(* IEC 61131-3 sources: eCockpitGit/test_project/src/%F%00 Library/%F%Common Functions/%F%String/%F%Big Input/%F%Concat, 9 files *)

(* ---- %POU%FU_sConcat10BI.st ---- *)
//This functions combines ten strings
//This is the big input version which means any size string can be inputted, but only string variables will be accepted
//It is also faster on bigger strings
// |**Version**|**Author**| **Date** |**Changes**
// | 1         | NSN      | 05-02-19 | Creation
// | 2         | NSN      | 14-10-21 | Changed to pointer based
FUNCTION FU_sConcat10BI : STRING(255)
VAR_INPUT
	s1			:POINTER TO EASCII;			//Input String1
	s2			:POINTER TO EASCII;			//Input String2
	s3			:POINTER TO EASCII;			//Input String3
	s4			:POINTER TO EASCII;			//Input String4
	s5			:POINTER TO EASCII;			//Input String5
	s6			:POINTER TO EASCII;			//Input String6
	s7			:POINTER TO EASCII;			//Input String7
	s8			:POINTER TO EASCII;			//Input String8
	s9			:POINTER TO EASCII;			//Input String9
	s10			:POINTER TO EASCII;			//Input String10
END_VAR
(*%!%__DELIMITER__%!%*)
FU_sConcat10BIBO(sOut:=ADR(FU_sConcat10BI),s1:=s1,s2:=s2,s3:=s3,s4:=s4,s5:=s5,s6:=s6,s7:=s7,s8:=s8,s9:=s9,s10:=s10,wOutSize:=255);

(* ---- %POU%FU_sConcat3BI.st ---- *)
//This functions combines three strings
//This is the big input version which means any size string can be inputted, but only string variables will be accepted
//It is also faster on bigger strings
// |**Version**|**Author**| **Date** |**Changes**
// | 1         | NSN      | 05-02-19 | Creation
// | 2         | NSN      | 14-10-21 | Changed to pointer based
FUNCTION FU_sConcat3BI : STRING(255)
VAR_INPUT
	s1			:POINTER TO EASCII;						//Input String1
	s2			:POINTER TO EASCII;						//Input String2
	s3			:POINTER TO EASCII;						//Input String3
END_VAR
(*%!%__DELIMITER__%!%*)
FU_sConcat3BIBO(sOut:=ADR(FU_sConcat3BI),s1:=s1,s2:=s2,s3:=s3,wOutSize:=255);

(* ---- %POU%FU_sConcat4BI.st ---- *)
//This functions combines four strings
//This is the big input version which means any size string can be inputted, but only string variables will be accepted
//It is also faster on bigger strings
// |**Version**|**Author**| **Date** |**Changes**
// | 1         | NSN      | 05-02-19 | Creation
// | 2         | NSN      | 14-10-21 | Changed to pointer based
FUNCTION FU_sConcat4BI : STRING(255)
VAR_INPUT
	s1			:POINTER TO EASCII;			//Input String1
	s2			:POINTER TO EASCII;			//Input String2
	s3			:POINTER TO EASCII;			//Input String3
	s4			:POINTER TO EASCII;			//Input String4
END_VAR
(*%!%__DELIMITER__%!%*)
FU_sConcat4BIBO(sOut:=ADR(FU_sConcat4BI),s1:=s1,s2:=s2,s3:=s3,s4:=s4,wOutSize:=255);

(* ---- %POU%FU_sConcat5BI.st ---- *)
//This functions combines five strings
//This is the big input version which means any size string can be inputted, but only string variables will be accepted
//It is also faster on bigger strings
// |**Version**|**Author**| **Date** |**Changes**
// | 1         | NSN      | 05-02-19 | Creation
// | 2         | NSN      | 14-10-21 | Changed to pointer based
FUNCTION FU_sConcat5BI : STRING(255)
VAR_INPUT
	s1			:POINTER TO EASCII;			//Input String1
	s2			:POINTER TO EASCII;			//Input String2
	s3			:POINTER TO EASCII;			//Input String3
	s4			:POINTER TO EASCII;			//Input String4
	s5			:POINTER TO EASCII;			//Input String5
END_VAR
(*%!%__DELIMITER__%!%*)
FU_sConcat5BIBO(sOut:=ADR(FU_sConcat5BI),s1:=s1,s2:=s2,s3:=s3,s4:=s4,s5:=s5,wOutSize:=255);

(* ---- %POU%FU_sConcat6BI.st ---- *)
//This functions combines six strings
//This is the big input version which means any size string can be inputted, but only string variables will be accepted
//It is also faster on bigger strings
// |**Version**|**Author**| **Date** |**Changes**
// | 1         | NSN      | 05-02-19 | Creation
// | 2         | NSN      | 14-10-21 | Changed to pointer based
FUNCTION FU_sConcat6BI : STRING(255)
VAR_INPUT
	s1			:POINTER TO EASCII;			//Input String1
	s2			:POINTER TO EASCII;			//Input String2
	s3			:POINTER TO EASCII;			//Input String3
	s4			:POINTER TO EASCII;			//Input String4
	s5			:POINTER TO EASCII;			//Input String5
	s6			:POINTER TO EASCII;			//Input String6
END_VAR
(*%!%__DELIMITER__%!%*)
FU_sConcat6BIBO(sOut:=ADR(FU_sConcat6BI),s1:=s1,s2:=s2,s3:=s3,s4:=s4,s5:=s5,s6:=s6,wOutSize:=255);

(* ---- %POU%FU_sConcat7BI.st ---- *)
//This functions combines seven strings
//This is the big input version which means any size string can be inputted, but only string variables will be accepted
//It is also faster on bigger strings
// |**Version**|**Author**| **Date** |**Changes**
// | 1         | NSN      | 05-02-19 | Creation
// | 2         | NSN      | 14-10-21 | Changed to pointer based
FUNCTION FU_sConcat7BI : STRING(255)
VAR_INPUT
	s1			:POINTER TO EASCII;			//Input String1
	s2			:POINTER TO EASCII;			//Input String2
	s3			:POINTER TO EASCII;			//Input String3
	s4			:POINTER TO EASCII;			//Input String4
	s5			:POINTER TO EASCII;			//Input String5
	s6			:POINTER TO EASCII;			//Input String6
	s7			:POINTER TO EASCII;			//Input String7
END_VAR
(*%!%__DELIMITER__%!%*)
FU_sConcat7BIBO(sOut:=ADR(FU_sConcat7BI),s1:=s1,s2:=s2,s3:=s3,s4:=s4,s5:=s5,s6:=s6,s7:=s7,wOutSize:=255);

(* ---- %POU%FU_sConcat8BI.st ---- *)
//This functions combines nine strings
//This is the big input version which means any size string can be inputted, but only string variables will be accepted
//It is also faster on bigger strings
// |**Version**|**Author**| **Date** |**Changes**
// | 1         | NSN      | 05-02-19 | Creation
// | 2         | NSN      | 14-10-21 | Changed to pointer based
FUNCTION FU_sConcat8BI : STRING(255)
VAR_INPUT
	s1			:POINTER TO EASCII;			//Input String1
	s2			:POINTER TO EASCII;			//Input String2
	s3			:POINTER TO EASCII;			//Input String3
	s4			:POINTER TO EASCII;			//Input String4
	s5			:POINTER TO EASCII;			//Input String5
	s6			:POINTER TO EASCII;			//Input String6
	s7			:POINTER TO EASCII;			//Input String7
	s8			:POINTER TO EASCII;			//Input String8
END_VAR
(*%!%__DELIMITER__%!%*)
FU_sConcat8BIBO(sOut:=ADR(FU_sConcat8BI),s1:=s1,s2:=s2,s3:=s3,s4:=s4,s5:=s5,s6:=s6,s7:=s7,s8:=s8,wOutSize:=255);

(* ---- %POU%FU_sConcat9BI.st ---- *)
//This functions combines nine strings
//This is the big input version which means any size string can be inputted, but only string variables will be accepted
//It is also faster on bigger strings
// |**Version**|**Author**| **Date** |**Changes**
// | 1         | NSN      | 05-02-19 | Creation
// | 2         | NSN      | 14-10-21 | Changed to pointer based
FUNCTION FU_sConcat9BI : STRING(255)
VAR_INPUT
	s1			:POINTER TO EASCII;			//Input String1
	s2			:POINTER TO EASCII;			//Input String2
	s3			:POINTER TO EASCII;			//Input String3
	s4			:POINTER TO EASCII;			//Input String4
	s5			:POINTER TO EASCII;			//Input String5
	s6			:POINTER TO EASCII;			//Input String6
	s7			:POINTER TO EASCII;			//Input String7
	s8			:POINTER TO EASCII;			//Input String8
	s9			:POINTER TO EASCII;			//Input String9
END_VAR
(*%!%__DELIMITER__%!%*)
FU_sConcat9BIBO(sOut:=ADR(FU_sConcat9BI),s1:=s1,s2:=s2,s3:=s3,s4:=s4,s5:=s5,s6:=s6,s7:=s7,s8:=s8,s9:=s9,wOutSize:=255);

(* ---- %POU%FU_sConcatBI.st ---- *)
//This functions combines two strings
//This is the big input version which means any size string can be inputted, but only string variables will be accepted
//It is also faster on bigger strings
// |**Version**|**Author**| **Date** |**Changes**
// | 1         | NSN      | 05-02-19 | Creation
// | 2         | NSN      | 14-10-21 | Changed to pointer based
FUNCTION FU_sConcatBI : STRING(255)
VAR_INPUT
	s1			:POINTER TO EASCII;			//Input String1
	s2			:POINTER TO EASCII;			//Input String2
END_VAR
(*%!%__DELIMITER__%!%*)
FU_sConcatBIBO(sOut:=ADR(FU_sConcatBI),s1:=s1,s2:=s2,wOutSize:=255);
